FUNCTION putString : bool
	VAR_INPUT
		stringPtr : POINTER TO STRING;
		stringLength : UINT;
	END_VAR
	VAR_IN_OUT
		bufferRef : POINTER TO USINT;
	END_VAR

	memcpy(bufferRef, stringPtr, stringLength);
	bufferRef := bufferRef + stringLength;
	putString := TRUE;

END_FUNCTION

(* stored: Version 1.1.0.1, ProductVersion 3.1.4024.3
   POU putString: Id {0cd1e89a-a6dd-0fab-12fb-b646f3ccf651}, SpecialFunc None *)
